TYPE Motion_Parameters_Type  :
STRUCT
	
	maxVelocity					: 		LREAL	:= 150;			// mm/s
	
	RotationScailing			: 		LREAL 	:= 0.0002; 		// 
	
	
END_STRUCT
END_TYPE

(* stored: Version 1.1.0.1, ProductVersion 3.1.4024.12
   DUT Motion_Parameters_Type: Id {d0b17dee-7333-45e8-9b59-4b5556caf9cf} *)
